// TwinCAT 3 PLC project TcoAbstractions
// Title: TcoAbstractions
// Company: Vortex.Library
// ProjectVersion: 0.6.0.913
// ProgramVersion: 3.1.4023.0
// libraries:
//   Tc2_Standard, * (Beckhoff Automation GmbH)
//   Tc2_System, * (Beckhoff Automation GmbH)
//   Tc3_Module, * (Beckhoff Automation GmbH)
//   TcoCore, 0.6.0.913 (Vortex.Library)
// project tree:
//   / PlcTask.TcTTO
//   Robotics/ CoordinatesAreEqual.TcPOU, eTcoRoboticsStopType.TcDUT, CalculateDistance.TcPOU, eTcoRoboticsDistance.TcDUT, IsNearlyEqual.TcPOU, ITcoRobotics.TcIO, TcoRoboticsCoordinates.TcDUT, TcoRoboticsBasicCoordinates.TcDUT, TcoRoboticsMovementsParams.TcDUT
//   Vision/CodeReader/ ITcoCodeReader.TcIO
// real-time tasks:
//   TASK PlcTask: cycle T#10ms, priority 20, ADS port 350
//   TASK PlcTask1: cycle T#10ms, priority 21, ADS port 351

CONFIGURATION TcoAbstractions
    RESOURCE PLC ON TwinCAT3
        TASK PlcTask(INTERVAL := T#10ms, PRIORITY := 20);
    END_RESOURCE
END_CONFIGURATION

// ---- Robotics/eTcoRoboticsStopType.TcDUT
{attribute 'qualified_only'}
{attribute 'strict'}
TYPE eTcoRoboticsStopType :
(
    Soft := 10,
    Quick := 20
);
END_TYPE

// ---- Robotics/eTcoRoboticsDistance.TcDUT
TYPE eTcoRoboticsDistance :
(
    X := 1,
    Y := 2,
    Z := 3,
    XY := 4,
    XZ := 5,
    YZ := 6,
    XYZ := 7
);
END_TYPE

// ---- Robotics/TcoRoboticsCoordinates.TcDUT
TYPE TcoRoboticsCoordinates :
STRUCT
    {attribute  addProperty Name "<#Coordinate X#>"}
    X : REAL;
    {attribute  addProperty Name "<#Coordinate Y#>"}
    Y : REAL;
    {attribute  addProperty Name "<#Coordinate Z#>"}
    Z : REAL;
    {attribute  addProperty Name "<#Coordinate Rx#>"}
    Rx : REAL;
    {attribute  addProperty Name "<#Coordinate Ry#>"}
    Ry : REAL;
    {attribute  addProperty Name "<#Coordinate Rz#>"}
    Rz : REAL;
END_STRUCT
END_TYPE

// ---- Robotics/TcoRoboticsBasicCoordinates.TcDUT
TYPE TcoRoboticsBasicCoordinates :
STRUCT
    {attribute  addProperty Name "<#Coordinate X#>"}
    X : REAL;
    {attribute  addProperty Name "<#Coordinate Y#>"}
    Y : REAL;
    {attribute  addProperty Name "<#Coordinate Z#>"}
    Z : REAL;
END_STRUCT
END_TYPE

// ---- Robotics/TcoRoboticsMovementsParams.TcDUT
TYPE TcoRoboticsMovementsParams :
STRUCT
    {attribute addProperty Name "<#ActionNo#>"}
    ActionNo : BYTE;
    {attribute addProperty Name "<#GlobalSpeed#>"}
    GlobalSpeed : BYTE;
    {attribute addProperty Name "<#ToolNo#>"}
    ToolNo : BYTE;
    {attribute addProperty Name "<#WorkobjectNo#>"}
    WorkobjectNo : BYTE;
    {attribute addProperty Name "<#PointNo#>"}
    PointNo : BYTE;
    {attribute addProperty Name "<#UserSpecSpeed1#>"}
    UserSpecSpeed1 : INT;
    {attribute addProperty Name "<#UserSpecSpeed2#>"}
    UserSpecSpeed2 : INT;
    {attribute  addProperty Name "<#Coordinates#>"}
    Coordinates : TcoRoboticsCoordinates;
END_STRUCT
END_TYPE

// ---- Robotics/ITcoRobotics.TcIO
INTERFACE ITcoRobotics EXTENDS __System.IQueryInterface

METHOD StartAtMain : TcoCore.ITcoTaskStatus
END_METHOD

METHOD StartMotorsAndProgram : TcoCore.ITcoTaskStatus
END_METHOD

METHOD StartMovements : TcoCore.ITcoTaskStatus
VAR_INPUT
	inData : TcoRoboticsMovementsParams;
END_VAR
END_METHOD

METHOD StopMovements : TcoCore.ITcoTaskStatus
VAR_INPUT
	inStopType : eTcoRoboticsStopType;
END_VAR
END_METHOD

METHOD StopMovementsAndProgram : TcoCore.ITcoTaskStatus
VAR_INPUT
	inStopType : eTcoRoboticsStopType;
END_VAR
END_METHOD

END_INTERFACE

// ---- Vision/CodeReader/ITcoCodeReader.TcIO
INTERFACE ITcoCodeReader EXTENDS __System.IQueryInterface

METHOD ClearResultData : TcoCore.ITcoTaskStatus
END_METHOD

METHOD Read : TcoCore.ITcoTaskStatus
END_METHOD

END_INTERFACE

// ---- Robotics/CoordinatesAreEqual.TcPOU
FUNCTION CoordinatesAreEqual : bool
VAR_INPUT
    Coordinates1 : TcoRoboticsCoordinates;
    Coordinates2 : TcoRoboticsCoordinates;
    EpsilonX : REAL;
    EpsilonY : REAL;
    EpsilonZ : REAL;
    EpsilonRx : REAL;
    EpsilonRy : REAL;
    EpsilonRz : REAL;
END_VAR
VAR
END_VAR

CoordinatesAreEqual := IsNearlyEqual(Coordinates1.X, Coordinates2.X, EpsilonX) AND
    IsNearlyEqual(Coordinates1.Y, Coordinates2.Y, EpsilonY) AND
    IsNearlyEqual(Coordinates1.Z, Coordinates2.Z, EpsilonZ) AND
    IsNearlyEqual(Coordinates1.Rx, Coordinates2.Rx, EpsilonRx) AND
    IsNearlyEqual(Coordinates1.Ry, Coordinates2.Ry, EpsilonRy) AND
    IsNearlyEqual(Coordinates1.Rz, Coordinates2.Rz, EpsilonRz);

END_FUNCTION

// ---- Robotics/IsNearlyEqual.TcPOU
FUNCTION IsNearlyEqual : bool
VAR_INPUT
    Coordinate1 : REAL;
    Coordinate2 : REAL;
    Epsilon : REAL;
END_VAR
VAR
    AbsCoordinate1 : REAL;
    AbsCoordinate2 : REAL;
    Diff : REAL;
    Denominator : LREAL;
END_VAR

IsNearlyEqual := FALSE;
AbsCoordinate1 := ABS(Coordinate1);
AbsCoordinate2 := ABS(Coordinate2);
Diff := ABS(Coordinate1 - Coordinate2);
Denominator := AbsCoordinate1;
Denominator := Denominator + AbsCoordinate2;

IF Epsilon < 0 THEN
    RETURN;
END_IF

IF Coordinate1 = Coordinate2 THEN
    IsNearlyEqual := TRUE;
ELSIF (Coordinate1 = 0 OR Coordinate2 = 0) AND Diff <= Epsilon THEN
    IsNearlyEqual := Diff <= Epsilon;
ELSE
    IsNearlyEqual := Diff / Denominator <= Epsilon;
END_IF;

END_FUNCTION

// ---- Robotics/CalculateDistance.TcPOU
FUNCTION CalculateDistance : REAL
VAR_INPUT
    inDistType : eTcoRoboticsDistance;
    inP1 : TcoRoboticsCoordinates;
    inP2 : TcoRoboticsCoordinates;
END_VAR

CASE inDistType OF
    eTcoRoboticsDistance.X:
        CalculateDistance := SQRT(EXPT((inP1.X - inP2.X), 2));
    eTcoRoboticsDistance.Y:
        CalculateDistance := SQRT(EXPT((inP1.Y - inP2.Y), 2));
    eTcoRoboticsDistance.Z:
        CalculateDistance := SQRT(EXPT((inP1.Z - inP2.Z), 2));
    eTcoRoboticsDistance.XY:
        CalculateDistance := SQRT(EXPT((inP1.X - inP2.X), 2) + EXPT((inP1.Y - inP2.Y), 2));
    eTcoRoboticsDistance.XZ:
        CalculateDistance := SQRT(EXPT((inP1.X - inP2.X), 2) + EXPT((inP1.Z - inP2.Z), 2));
    eTcoRoboticsDistance.YZ:
        CalculateDistance := SQRT(EXPT((inP1.Y - inP2.Y), 2) + EXPT((inP1.Z - inP2.Z), 2));
    eTcoRoboticsDistance.XYZ:
        CalculateDistance := SQRT(EXPT((inP1.X - inP2.X), 2) + EXPT((inP1.Y - inP2.Y), 2) + EXPT((inP1.Z - inP2.Z), 2));
END_CASE

END_FUNCTION
